TEXTLIST E_MODE
  0 = 'IDLE'
  2 = 'MANUAL'
  1 = 'AUTOMATIC'
   = ''
END_TEXTLIST

(* stored: Version 1.1.0.1, ProductVersion 3.1.4024.12
   TextList E_MODE: Id {42a64ff1-3632-42e5-970d-8c06a20be4a2} *)
